Universal Robots PolyScope program: check get actual tcp pose.urp

Program check get actual tcp pose (installation=default directory=/programs createdIn=5.21.3 lastSavedIn=5.21.3 robotSerialNumber=20246801938)
Calibrated DH parameters: a=[-0.000071, -0.790281, -0.600694, 0.000061, -0.000039, 0]; d=[0.236272, 604.465945, 132.116513, -736.382239, 0.159268, 0.154005]; alpha=[1.570254, -0.000567, 0.000559, 1.571709, -1.56999, 0]; deltaTheta=[0, -0.409357, 7.293326, -0.600784, -0.000001, -0.000001]
InitVariablesNode
Robot Program (runOnlyOnce=true)
  var_1 := get_actual_tcp_pose()
  MoveL speed 250 mm/s, acceleration 1200 mm/s^2 (useActiveTCP=true optimoveEnabled=false optiMoveSpeed=0.3 optiMoveAcceleration=0.09) feature=Base
    MoveDirectionNode (selectedDirection=XPlus)
      Until DISTANCE (allowActions=false deceleration=3 distanceNodeType=STOP) Distance=0.1; motionParameters(blendRadius=0)
  Set NoAction tcp=TCP
  Set NoAction tcp=pretend_w_top
  MoveJ speed 60 deg/s, acceleration 80 deg/s^2 (useActiveTCP=true optimoveEnabled=false optiMoveSpeed=0.3 optiMoveAcceleration=0.09) feature=Base
    Waypoint Variable (Variable): variable=var_1
